PROGRAM GitHub1
VAR
	Testi100	: INT;
	Testi101	: BOOL;
	Testi102	: INT;	
END_VAR

IF Testi101 THEN
	Testi100 := Testi100 + 2;
END_IF

END_PROGRAM

(* stored: Version 1.1.0.1, ProductVersion 3.1.4024.12
   POU GitHub1: Id {4130db12-1102-4508-b046-e234a13b982b}, SpecialFunc None *)
